FUNCTION_BLOCK FB_WrappedMembers
VAR_INPUT
    bEnable : BOOL;
    sLabel  : STRING;
END_VAR
VAR_OUTPUT
    sStatus : STRING;
END_VAR
VAR
    nRuns : UINT;
END_VAR

IF bEnable THEN
    sStatus := CONCAT(sLabel, ' active');
ELSE
    sStatus := CONCAT(sLabel, ' idle');
END_IF;

PROPERTY Status : STRING
END_PROPERTY

METHOD Start : BOOL
IF bEnable THEN
    nRuns := nRuns + 1;
    Start := TRUE;
ELSE
    Start := FALSE;
END_IF;
END_METHOD

METHOD Stop : BOOL
Stop := nRuns > 0;
END_METHOD

ACTION Refresh:
sStatus := CONCAT(sLabel, ' refreshed');
END_ACTION

END_FUNCTION_BLOCK

(* stored: Version 1.1.0.1, ProductVersion 3.1.4024.10
   POU FB_WrappedMembers: KindOfPOU Element
   Method Start: KindOfMethod Element
   Method Stop: KindOfMethod Element
   Action Refresh: KindOfAction Element *)
